// TIA Portal V20 export
// export: Created 2025-12-01T14:57:05.8674174Z, ExportSetting None, DisplayName Totally Integrated Automation Portal, DisplayVersion V20 Update 3, DisplayName TIA Portal Openness, DisplayVersion V20 Update 3, DisplayName TIA Portal Version Control Interface, DisplayVersion V20 Update 3, DisplayName STEP 7 Professional, DisplayVersion V20 Update 3, DisplayName STEP 7 Safety, DisplayVersion V20 Update 2, DisplayName WinCC Basic/Comfort/Advanced, DisplayVersion V20 Update 3, DisplayName WinCC Professional, DisplayVersion V20 Update 3, DisplayName WinCC Unified, DisplayVersion V20 Update 3
FUNCTION "FC891_EtiqDInt_EtiqChar" : Void   // FC891, LAD
{ S7_Optimized_Access := 'FALSE' }
AUTHOR : TRACKING
NAME : 20130301
VERSION : 3.0
// stored: AutoNumber false, SetENOAutomatically false
   VAR_INPUT
      DB_String : UInt;
      Long_String : UInt;
      Offset_Ini : UInt;   // Apunta al Caracter de menor peso del Entero representado en el String
      Valor : UDInt;
   END_VAR
   VAR_TEMP
      puntero_CHAR : DWord;
      N_DB : Word;
      CNT_Caracteres : UInt;
      Offset_Actual : UInt;
      Peso_Caracter : UDInt;
      Valor_Caracter : UInt;
      Valor_Restante : UDInt;
   END_VAR
BEGIN

NETWORK
TITLE = 
      L     #DB_String;
      T     #N_DB;
//==================================
      L     0;
      T     #CNT_Caracteres;  //Inicializa el contador de caracteres de Lectura
//==================================
      L     #Offset_Ini;  // Pasa el dato del Offset inicial a una variable de Trabajo
      T     #Offset_Actual;
//===================================
      L     #Valor;  //Inicia el valor de la función
      T     #Valor_Restante;

NETWORK
TITLE = 
      OPN   DB [#N_DB];

BUCLE:L     #Offset_Actual;  //Obtener direccion actual del caractera a tratar en el db
      SLD   3;  //Dar formato de Integer a Puntero
      T     #puntero_CHAR;  //Guardamos Puntero a Caracter en DB
//=================================
      L     #Valor_Restante;  //Validamos que se trata de un número> 0
      L     0;  //'0' caracter es el Hexadecimal 30
      <D;
      JC    FIN;
//=================================
      L     #Valor_Restante;
      L     10;
      MOD;
      L     W#16#30;
      +I;
      T     DBB [#puntero_CHAR];  //Eliminamos la parte alta del BYTE
//=================================
      L     #Valor_Restante;
      L     10;
      /D;
      T     #Valor_Restante;
//==================================
      L     #Offset_Actual;  //No posicionamos en el caracter anterior
      L     -1;
      +I;
      T     #Offset_Actual;
//==================================
      L     1;
      L     #CNT_Caracteres;  //Incrementa el contador de caracteres
      +I;
      T     #CNT_Caracteres;
      L     #Long_String;
      <I;
      JC    BUCLE;
//==================================

FIN:  NOP   0;
END_FUNCTION
